// Mitsubishi GX Works2 project: 더하기   PLC: Q02/Q02H

PROGRAM MAIN
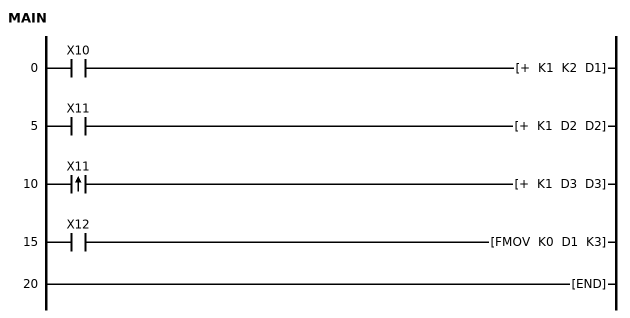
0     LD      X10
      +       K1 K2 D1
5     LD      X11
      +       K1 D2 D2
10    LDP     X11
      +       K1 D3 D3
15    LD      X12
      FMOV    K0 D1 K3
20    END
END_PROGRAM
